INTERFACE ITcoInputDialogAnswer EXTENDS ITcoInputDialogFormat

PROPERTY Answer : eInputDialogAnswer
GET
END_GET
END_PROPERTY

END_INTERFACE

(* stored: Version 1.1.0.1
   Itf ITcoInputDialogAnswer: Id {0a757a56-ddf8-0a00-24fc-0d95df792179}
   Property Answer: Id {ed328233-290c-0717-3b5b-c1190568855d}
   Get Get: Id {11e8414b-bbd9-0b00-1b71-a25c17c6b3a9} *)
